{attribute 'qualified_only'}
{attribute 'strict'}
TYPE E_ForceValue :
(
	RELEASED := 0,
	FORCE_ON := 1,
	FORCE_OFF := 2
);
END_TYPE

(* stored: Version 1.1.0.1, ProductVersion 3.1.4024.12
   DUT E_ForceValue: Id {2af6e411-0eb9-4cfc-89e1-adcfe0348636} *)
